{attribute 'linkalways'} 
{attribute 'no_explicit_call' := 'This FB is a CLASS and must be accessed using methods or properties'}
{attribute 'enable_dynamic_creation'}
FUNCTION_BLOCK FINAL AND_UINT EXTENDS Node
VAR
	in1 : _UINT(0);
	in2 : _UINT(0);
	out : _UINT(0);
END_VAR

METHOD PUBLIC Clone : I_Node
VAR
	pNode : POINTER TO AND_UINT;
END_VAR
pNode := __NEW(AND_UINT);
Clone := pNode^;
END_METHOD

METHOD FB_init : BOOL
VAR_INPUT
	bInitRetains : BOOL; // if TRUE, the retain variables are initialized (warm start / cold start)
	bInCopyCode : BOOL;  // if TRUE, the instance afterwards gets moved into the copy code (online change)
END_VAR
AddInput('in1',THIS^.in1);
AddInput('in2',THIS^.in2);
AddOutput('out', THIS^.out);
END_METHOD

METHOD PROTECTED OnExecute
VAR
END_VAR
out.Value := in1.Value AND in2.Value;
END_METHOD

END_FUNCTION_BLOCK

(* stored: Version 1.1.0.1, ProductVersion 3.1.4024.15
   POU AND_UINT: Id {b8b74403-1fa2-48d0-9b85-1883e1f91ced}, SpecialFunc None
   Folder Constructor: Id {fd7efcaa-a6ca-4fa4-8150-ec852792a0a6}
   Method Clone: Id {a2ecb9ae-9b34-41e2-9727-43b367a41729}
   Method FB_init: Id {00e4ccd6-221c-4b21-9a40-f3936f471815}
   Method OnExecute: Id {20a628fe-b031-4dd4-99e4-f5c127529017} *)
